// TIA Portal V18 program export: 1 tag tables, 0 data types, 0 data blocks, 2 code blocks (in call order from the OBs), 1 instance data blocks

VAR_GLOBAL   // PLC tag table "Default tag table"
   FlowOn AT %Q0.1 : Bool;
   RemoteOnCommand AT %I0.1 : Bool;
END_VAR

ORGANIZATION_BLOCK "Main"   // OB1, LAD, ProgramCycle
TITLE = "Main Program Sweep (Cycle)"
{ S7_Optimized_Access := 'TRUE' }
VERSION : 0.1
// stored: AutoNumber true, IsIECCheckEnabled false, SetENOAutomatically false
BEGIN

REGION Network 1
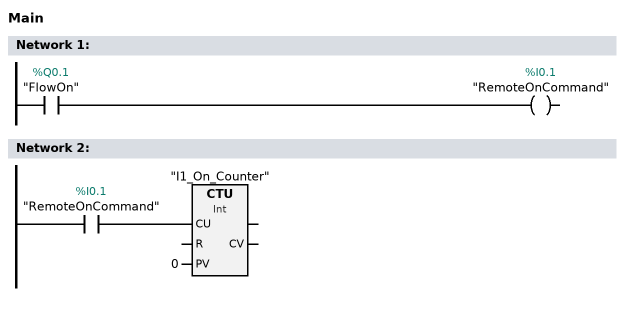
   RUNG wire#powerrail
      Contact( "FlowOn" )
      Coil( "RemoteOnCommand" )
   END_RUNG
   // the same network as SCL:
   "RemoteOnCommand" := "FlowOn";
END_REGION

REGION Network 2
   RUNG wire#powerrail
      Contact( "RemoteOnCommand" )
      { S7_Templates := "value_type := Int" } "I1_On_Counter".CTU(r :=, pv := 0, cv =>)
   END_RUNG
   // the same network as SCL:
   "I1_On_Counter".CTU(CU := "RemoteOnCommand", PV := 0);
END_REGION
END_ORGANIZATION_BLOCK

ORGANIZATION_BLOCK "Startup"   // OB100, LAD, Startup
TITLE = "Complete Restart"
{ S7_Optimized_Access := 'TRUE' }
VERSION : 0.1
// stored: AutoNumber true, IsIECCheckEnabled false, SetENOAutomatically false
   VAR_INPUT
      LostRetentive : Bool;   // True if retentive data are lost
      LostRTC : Bool;   // True if date and time are lost
   END_VAR
BEGIN

REGION Network 1
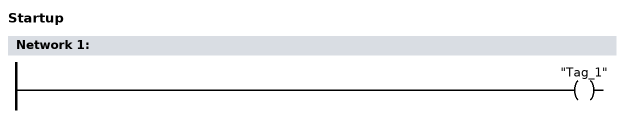
   RUNG wire#powerrail
      Coil( "Tag_1" )
   END_RUNG
   // the same network as SCL:
   "Tag_1" := TRUE;
END_REGION
END_ORGANIZATION_BLOCK

DATA_BLOCK "I1_On_Counter"   // DB1
{ S7_Optimized_Access := 'TRUE' }
// stored: AutoNumber false, InstanceOfName IEC_COUNTER, OfSystemLibElement IEC_COUNTER, OfSystemLibVersion 1.0
"IEC_COUNTER"
   // VAR RETAIN
   //    CU : Bool;
   //    CD : Bool;
   //    R : Bool;
   //    LD : Bool;
   //    QU : Bool;
   //    QD : Bool;
   //    PV : Int;
   //    CV : Int;
   // END_VAR
BEGIN
END_DATA_BLOCK
